{attribute 'qualified_only'}
{attribute 'strict'}
TYPE E_HomingState :
(
	Idle			:= 0,
	FirstHoming		:= 1,
	Reverse			:= 11,
	Inverse			:= 12,
	Re				:= 2,
	SecondHoming	:= 3,
	Done			:= 4
) := Idle;
END_TYPE

(* stored: Version 1.1.0.1, ProductVersion 3.1.4024.12
   DUT E_HomingState: Id {46dcca8c-b5a3-4d10-8c2c-84e0ab9c23ef} *)
